{attribute 'qualified_only'}
VAR_GLOBAL
END_VAR

(* stored: Version 1.1.0.1, ProductVersion 3.1.4024.11
   GVL G_Safety: Id {46833ddd-2c31-4feb-ba64-c15012a97589} *)
